# EPICS substitutions: bsaDriverApp/Db/bsas.substitutions
file bsasChannelCtrl.db {
    pattern {   DEVICE    }
            {   "$(DEV)"  }
}
